// TIA Portal V20 export
DATA_BLOCK "IdentRfHmi"   // DB213
// stored: MemoryReserve 100
   VAR
      IdentRf : Array[0.."NO_OF_RF_IDENT_DEVICES"] of "typeIdentRf";
      MobileRFID : "LER_typeMobileRFIDInterface";
   END_VAR
BEGIN
END_DATA_BLOCK
